FUNCTION_BLOCK L0_IncomEx (* Basic Function Block Type *)
  (* Standard: 61499-2 *)
  (* Version 0.0, 2014-09-04, 4DIAC-IDE, 4DIAC-Consortium *)
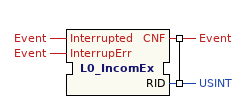
  EVENT_INPUT
    Interrupted; (* CNC Interrupted event *)
    InterrupErr; (* CNC Interrupted by Error *)
  END_EVENT
  EVENT_OUTPUT
    CNF WITH RID; (* Execution Confirmation *)
  END_EVENT
  VAR_OUTPUT
    RID : USINT; (* Error return ID *)
  END_VAR
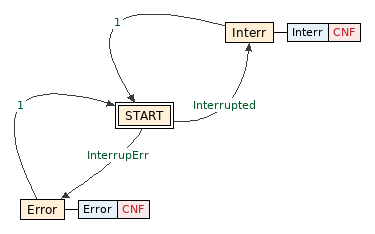
  EC_STATES
    START; (* Initial State *)
    Interr : Interr -> CNF; (* Initialization *)
    Error : Error -> CNF; (* Normal execution *)
  END_STATES
  EC_TRANSITIONS
    START TO Interr := Interrupted;
    Interr TO START := 1;
    START TO Error := InterrupErr;
    Error TO START := 1;
  END_TRANSITIONS
  ALGORITHM Interr IN ST: (* CNC Interrupted algo *)
RID := 1;
  END_ALGORITHM
  ALGORITHM Error IN ST: (* CNC interrupted by error algo *)
RID := 2;
  END_ALGORITHM
END_FUNCTION_BLOCK
